(* CODESYS project AutomatedWarehouse.project

Project tree, tasks and I/O mapping:
  Device : CODESYS Control Win V3 x64, CODESYS, version 3.5.22.20
    application Application
      libraries: Standard, 3.5.22.0 (System)
      task MainTask (cyclic, interval t#20ms, priority 1) calls PLC_PRG
      Symbols
      program PLC_PRG [?]
      global variables IO
    Ethernet : Ethernet, CODESYS, version 4.2.0.0
      ModbusTCP_Server_Device : ModbusTCP Server Device, CODESYS, version 4.5.0.0
          settings: DistinctBitAreas = TRUE; Coils Size = 15; Discrete Inputs Size = 10
          output Application.IO.Target_Position : WORD  // Input Registers.Input Registers
          input  Application.IO.At_Entry_Sensor : BOOL  // Coils.Coils.Bit0
          input  Application.IO.At_Load_Sensor : BOOL  // Coils.Coils.Bit1
          input  Application.IO.At_Left_Sensor : BOOL  // Coils.Coils.Bit2
          input  Application.IO.At_Middle_Sensor : BOOL  // Coils.Coils.Bit3
          input  Application.IO.At_Right_Sensor : BOOL  // Coils.Coils.Bit4
          input  Application.IO.At_Unload_Sensor : BOOL  // Coils.Coils.Bit5
          input  Application.IO.At_Exit_Sensor : BOOL  // Coils.Coils.Bit6
          input  Application.IO.Moving_X : BOOL  // Coils.Coils.Bit7
          input  Application.IO.Moving_Z : BOOL  // Coils.Coils.Bit0
          input  Application.IO.Start : BOOL  // Coils.Coils.Bit1
          input  Application.IO.Reset : BOOL  // Coils.Coils.Bit2
          input  Application.IO.Stop : BOOL  // Coils.Coils.Bit3
          input  Application.IO.Emergency_Stop : BOOL  // Coils.Coils.Bit4
          input  Application.IO.Mode_Unload : BOOL  // Coils.Coils.Bit5
          output Application.IO.Entry_Conveyor_CMD : BOOL  // Discrete Inputs.Discrete Inputs.Bit0
          output Application.IO.Load_Conveyor_CMD : BOOL  // Discrete Inputs.Discrete Inputs.Bit1
          output Application.IO.Forks_Left_CMD : BOOL  // Discrete Inputs.Discrete Inputs.Bit2
          output Application.IO.Forks_Right_CMD : BOOL  // Discrete Inputs.Discrete Inputs.Bit3
          output Application.IO.Lift_CMD : BOOL  // Discrete Inputs.Discrete Inputs.Bit4
          output Application.IO.Unload_Conveyor_CMD : BOOL  // Discrete Inputs.Discrete Inputs.Bit5
          output Application.IO.Exit_Conveyor_CMD : BOOL  // Discrete Inputs.Discrete Inputs.Bit6
          output Application.IO.Start_Status_Light : BOOL  // Discrete Inputs.Discrete Inputs.Bit7
          output Application.IO.Reset_Status_Light : BOOL  // Discrete Inputs.Discrete Inputs.Bit0
          output Application.IO.Stop_Status_Light : BOOL  // Discrete Inputs.Discrete Inputs.Bit1
          unmapped channels: Holding Registers, Input Registers, Coils, Discrete Inputs
*)

// Device/Application/IO
{attribute 'qualified_only'}
VAR_GLOBAL
	At_Entry_Sensor: BOOL;
	At_Load_Sensor: BOOL;
	Entry_Conveyor_CMD: BOOL;
	Load_Conveyor_CMD: BOOL;
	At_Left_Sensor: BOOL;
	At_Middle_Sensor: BOOL;
	At_Right_Sensor: BOOL;
	At_Unload_Sensor: BOOL;
	At_Exit_Sensor: BOOL;
	Moving_X: BOOL;
	Moving_Z: BOOL;
	Start: BOOL;
	Reset: BOOL;
	Stop: BOOL;
	Emergency_Stop: BOOL;
	Mode_Unload: BOOL;
	Forks_Left_CMD: BOOL;
	Forks_Right_CMD: BOOL;
	Lift_CMD: BOOL;
	Unload_Conveyor_CMD: BOOL;
	Exit_Conveyor_CMD: BOOL;
	Start_Status_Light: BOOL;
	Reset_Status_Light: BOOL;
	Stop_Status_Light: BOOL;
	Target_Position: INT;
END_VAR

// Device/Application/PLC_PRG
PROGRAM PLC_PRG

VAR
	Loading: BOOL;
	Receiving: BOOL;
	ReceivingDelayLift: TON;
	Transporting: BOOL;
	DelayAfterLift: TON;
	WaitForLeftForkRetract: TON;
	CurrentSlot: INT := 1;
	Storing: BOOL;
	CraneMoving: BOOL;
	StoringDelayLower: TON;
	DelayAfterLower: TON;
	Returning: BOOL;
	IncrementStorageCell: R_TRIG;
	DelayCraneReturnAfterRetract: TON;
	ReadyToStop: BOOL;
	RetrievingDelayLift: TON;
	DelayForkReturn: TON;
	Retrieving: BOOL;
	UnLoading: BOOL;
	ReturningUnload: BOOL;
	DelayCraneReturnAfterRetract2: TON;
	InPosition: BOOL;
	DecrementStorageCell: R_TRIG;
	SetRightForks: R_TRIG;
	DelayLowerUnload: TON;
	DelayRetractAfterLower: TON;
	UnloadConveyors: BOOL;
	Removed: BOOL;
	PulseConveyorTimer: TP;
	DelayUnloadConveyorReset: TON;
	PulseForkTimer: TP;
	ReadyToStart: BOOL;
	ResetStopBit: R_TRIG;
	DecrementStorageCellReset: R_TRIG;
END_VAR

(* body of a kind this reader does not render *)

END_PROGRAM
